// TIA Portal V19 export
FUNCTION "VFD Control" : Void   // FC9, LAD
{ S7_Optimized_Access := 'TRUE' }
// stored: SetENOAutomatically false
   VAR_TEMP   // added for the SCL form of the ladder/FBD networks
      _w1 : Bool;
   END_VAR
BEGIN

REGION Network 1: Liquids Pump
   // Refspeed = p2000, ref_Current = P2002, Ref_torque = P2003
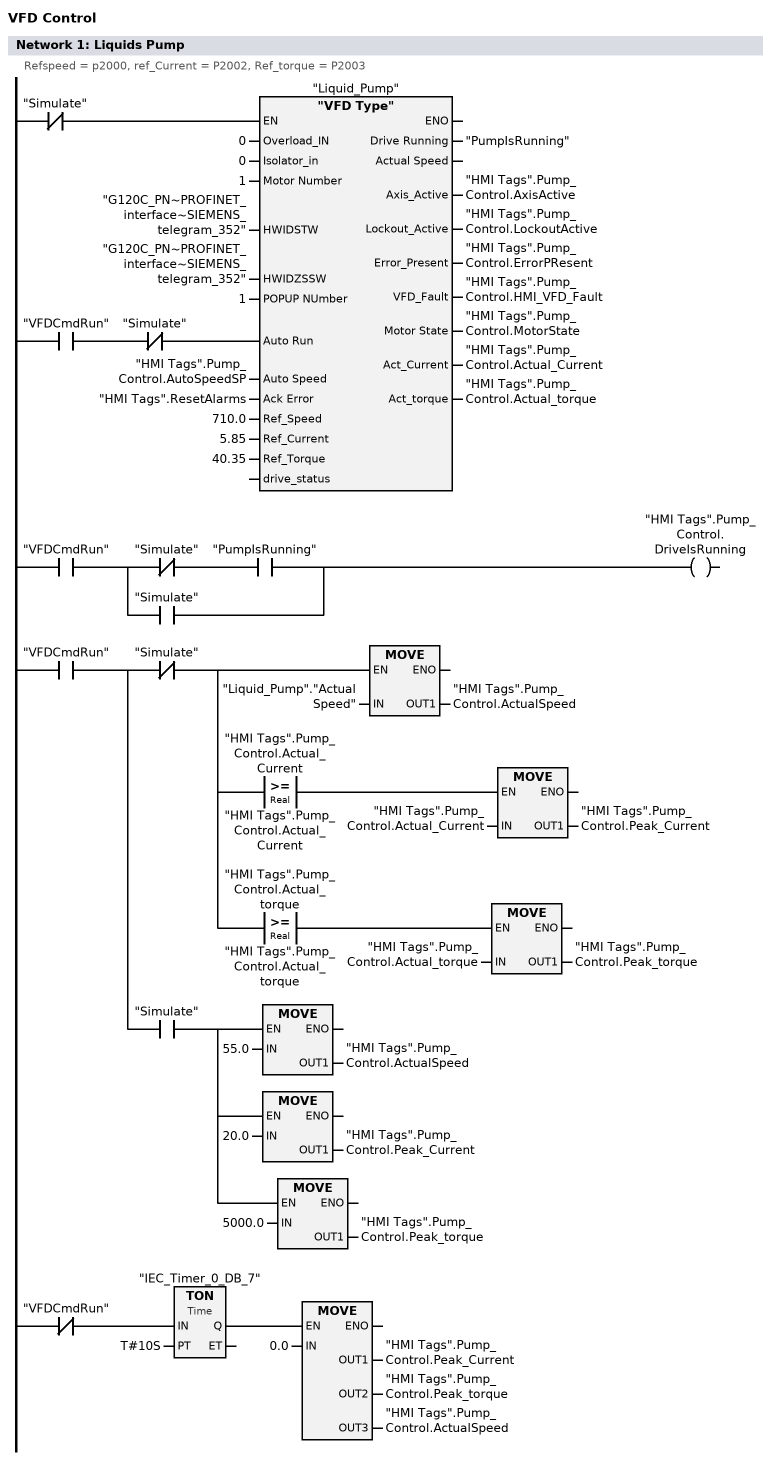
   RUNG wire#powerrail
      I_Contact( "Simulate" )
      "Liquid_Pump"("Auto Run" := wire#w1, Overload_IN := 0, Isolator_in := 0, "Motor Number" := 1, HWIDSTW := "G120C_PN~PROFINET_interface~SIEMENS_telegram_352", HWIDZSSW := "G120C_PN~PROFINET_interface~SIEMENS_telegram_352", "POPUP NUmber" := 1, "Auto Speed" := "HMI Tags".Pump_Control.AutoSpeedSP, "Ack Error" := "HMI Tags".ResetAlarms, Ref_Speed := 710.0, Ref_Current := 5.85, Ref_Torque := 40.35, drive_status :=, "Drive Running" => "PumpIsRunning", "Actual Speed" =>, Axis_Active => "HMI Tags".Pump_Control.AxisActive, Lockout_Active => "HMI Tags".Pump_Control.LockoutActive, Error_Present => "HMI Tags".Pump_Control.ErrorPResent, VFD_Fault => "HMI Tags".Pump_Control.HMI_VFD_Fault, "Motor State" => "HMI Tags".Pump_Control.MotorState, Act_Current => "HMI Tags".Pump_Control.Actual_Current, Act_torque => "HMI Tags".Pump_Control.Actual_torque)
   END_RUNG
   RUNG wire#powerrail
      Contact( "VFDCmdRun" )
      I_Contact( "Simulate" )
   END_RUNG wire#w1
   RUNG wire#powerrail
      Contact( "VFDCmdRun" )
      wire#w2
      I_Contact( "Simulate" )
      Contact( "PumpIsRunning" )
      wire#w3
      Coil( "HMI Tags".Pump_Control.DriveIsRunning )
   END_RUNG
   RUNG wire#w2
      Contact( "Simulate" )
   END_RUNG wire#w3
   RUNG wire#powerrail
      Contact( "VFDCmdRun" )
      wire#w4
      I_Contact( "Simulate" )
      wire#w5
      Move(in := "Liquid_Pump"."Actual Speed", out1 => "HMI Tags".Pump_Control.ActualSpeed)
   END_RUNG
   RUNG wire#w5
      { S7_Templates := "SrcType := Real" } GE_Contact(in1 := "HMI Tags".Pump_Control.Actual_Current, in2 := "HMI Tags".Pump_Control.Actual_Current)
      Move(in := "HMI Tags".Pump_Control.Actual_Current, out1 => "HMI Tags".Pump_Control.Peak_Current)
   END_RUNG
   RUNG wire#w5
      { S7_Templates := "SrcType := Real" } GE_Contact(in1 := "HMI Tags".Pump_Control.Actual_torque, in2 := "HMI Tags".Pump_Control.Actual_torque)
      Move(in := "HMI Tags".Pump_Control.Actual_torque, out1 => "HMI Tags".Pump_Control.Peak_torque)
   END_RUNG
   RUNG wire#w4
      Contact( "Simulate" )
      wire#w6
      Move(in := 55.0, out1 => "HMI Tags".Pump_Control.ActualSpeed)
   END_RUNG
   RUNG wire#w6
      Move(in := 20.0, out1 => "HMI Tags".Pump_Control.Peak_Current)
   END_RUNG
   RUNG wire#w6
      Move(in := 5000.0, out1 => "HMI Tags".Pump_Control.Peak_torque)
   END_RUNG
   RUNG wire#powerrail
      I_Contact( "VFDCmdRun" )
      { S7_Templates := "time_type := Time" } "IEC_Timer_0_DB_7".TON(pt := T#10S, et =>)
      Move(in := 0.0, out1 => "HMI Tags".Pump_Control.Peak_Current, out2 => "HMI Tags".Pump_Control.Peak_torque, out3 => "HMI Tags".Pump_Control.ActualSpeed)
   END_RUNG
   // the same network as SCL:
   IF NOT "Simulate" THEN
       "Liquid_Pump"(Overload_IN := 0,   // "VFD Type"
                     Isolator_in := 0,
                     "Motor Number" := 1,
                     HWIDSTW := "G120C_PN~PROFINET_interface~SIEMENS_telegram_352",
                     HWIDZSSW := "G120C_PN~PROFINET_interface~SIEMENS_telegram_352",
                     "POPUP NUmber" := 1,
                     "Auto Run" := "VFDCmdRun" AND NOT "Simulate",
                     "Auto Speed" := "HMI Tags".Pump_Control.AutoSpeedSP,
                     "Ack Error" := "HMI Tags".ResetAlarms,
                     Ref_Speed := 710.0,
                     Ref_Current := 5.85,
                     Ref_Torque := 40.35,
                     "Drive Running" => "PumpIsRunning",
                     Axis_Active => "HMI Tags".Pump_Control.AxisActive,
                     Lockout_Active => "HMI Tags".Pump_Control.LockoutActive,
                     Error_Present => "HMI Tags".Pump_Control.ErrorPResent,
                     VFD_Fault => "HMI Tags".Pump_Control.HMI_VFD_Fault,
                     "Motor State" => "HMI Tags".Pump_Control.MotorState,
                     Act_Current => "HMI Tags".Pump_Control.Actual_Current,
                     Act_torque => "HMI Tags".Pump_Control.Actual_torque);
   END_IF;
   "HMI Tags".Pump_Control.DriveIsRunning := "VFDCmdRun" AND ((NOT "Simulate" AND "PumpIsRunning") OR "Simulate");
   #_w1 := "VFDCmdRun" AND NOT "Simulate";
   IF #_w1 THEN "HMI Tags".Pump_Control.ActualSpeed := "Liquid_Pump"."Actual Speed"; END_IF;
   IF #_w1 AND ("HMI Tags".Pump_Control.Actual_Current >= "HMI Tags".Pump_Control.Actual_Current) THEN
       "HMI Tags".Pump_Control.Peak_Current := "HMI Tags".Pump_Control.Actual_Current;
   END_IF;
   IF #_w1 AND ("HMI Tags".Pump_Control.Actual_torque >= "HMI Tags".Pump_Control.Actual_torque) THEN
       "HMI Tags".Pump_Control.Peak_torque := "HMI Tags".Pump_Control.Actual_torque;
   END_IF;
   IF "VFDCmdRun" AND "Simulate" THEN
       "HMI Tags".Pump_Control.ActualSpeed := 55.0;
       "HMI Tags".Pump_Control.Peak_Current := 20.0;
       "HMI Tags".Pump_Control.Peak_torque := 5000.0;
   END_IF;
   "IEC_Timer_0_DB_7".TON(IN := NOT "VFDCmdRun", PT := T#10S);
   IF "IEC_Timer_0_DB_7".Q THEN
       "HMI Tags".Pump_Control.Peak_Current := 0.0;
       "HMI Tags".Pump_Control.Peak_torque := 0.0;
       "HMI Tags".Pump_Control.ActualSpeed := 0.0;
   END_IF;
END_REGION
END_FUNCTION
